Staubli VAL3: trimString.pgx

public program trimString(string& x_sInput[], string& x_sResult[])
  local num l_nLength
  local num l_nElement
  local string l_sLine
  local num l_nPos
begin

  l_nLength = size(x_sInput)
  resize(x_sResult,1,1)
  x_sResult = ""
  resize(x_sResult,1,l_nLength)

  for l_nElement = 0 to l_nLength-1

    // copy line
    l_sLine = x_sInput[l_nElement]

    while find(l_sLine," ")>=0
      l_nPos = find(l_sLine," ")
      l_sLine=delete(l_sLine,1,l_nPos)
    endWhile

    x_sResult[l_nElement] = l_sLine

  endFor

end
